// Mitsubishi GX Works2 project: PLC_Project_v156 final   PLC: FX3G

// global labels: Global1
VAR_GLOBAL
  X_0 AT X000 : BOOL;
  X_1 AT X001 : BOOL;
  X_2 AT X002 : BOOL;
  X_3 AT X003 : BOOL;
  X_4 AT X004 : BOOL;
  X_5 AT X005 : BOOL;
  X_6 AT X006 : BOOL;
  X_7 AT X007 : BOOL;
  Y_0 AT Y000 : BOOL;
  Y_1 AT Y001 : BOOL;
  Y_2 AT Y002 : BOOL;
  Y_3 AT Y003 : BOOL;
  Y_4 AT Y004 : BOOL;
  Y_5 AT Y005 : BOOL;
  Y_6 AT Y006 : BOOL;
  Y_7 AT Y007 : BOOL;
  SINGLE_POP_PACK : BOOL;
  FLVR_PRO_START : BOOL;
  COOLING_START : BOOL;
  TEMP_SENSOR : BOOL;
  PACKAGING_START : BOOL;
  EMERGENCY_BTN : BOOL;
  FACTORY_START : BOOL;
  FLVR_RUNNING : BOOL;
  COOLING_RUNNING : BOOL;
  CASE_PAC_RUNNING : BOOL;
  FACTORY_RUNNING : BOOL;
  ANALOG_1 AT D8280 : INT;
  TOTAL_BOX : INT;
  POP_COUNT AT CC1 : BOOL;
  COUNTER1 AT CC2 : BOOL;
  CN_1 AT CN1 : WORD;
  ANALOG_OUTPUT AT D8282 : INT;
  TIMER3_RUN : BOOL;
  MIXING_BLINK1 : BOOL;
  MIXING_BLINK2 : BOOL;
END_VAR

// task Task_01 (event TRUE, interval 0, priority 31): IO_MAP, MAIN

PROGRAM IO_MAP
(* structured ladder/FBD written out as ST: instructions are called as NAME(EN, inputs, outputs); _pN, _eN, _tN stand for wires *)
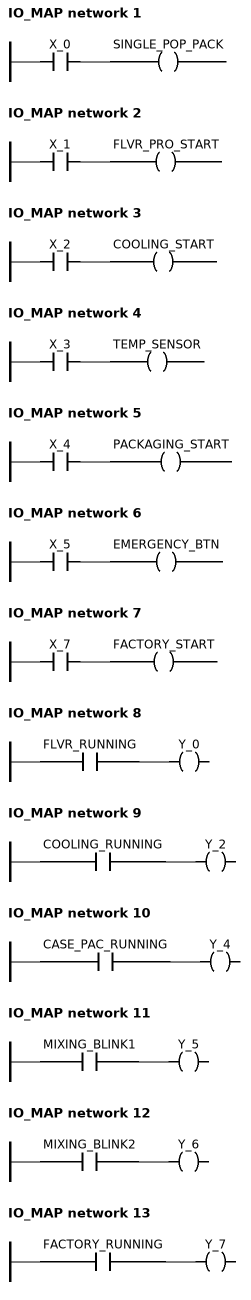
(* network 1 *)
SINGLE_POP_PACK := X_0;
(* network 2 *)
FLVR_PRO_START := X_1;
(* network 3 *)
COOLING_START := X_2;
(* network 4 *)
TEMP_SENSOR := X_3;
(* network 5 *)
PACKAGING_START := X_4;
(* network 6 *)
EMERGENCY_BTN := X_5;
(* network 7 *)
FACTORY_START := X_7;
(* network 8 *)
Y_0 := FLVR_RUNNING;
(* network 9 *)
Y_2 := COOLING_RUNNING;
(* network 10 *)
Y_4 := CASE_PAC_RUNNING;
(* network 11 *)
Y_5 := MIXING_BLINK1;
(* network 12 *)
Y_6 := MIXING_BLINK2;
(* network 13 *)
Y_7 := FACTORY_RUNNING;
END_PROGRAM

PROGRAM MAIN
VAR
  READY : BOOL;
  REGULAR_POP : BOOL;
  LARGE_POP : BOOL;
  POP_FLAVOR_SEL : BOOL;
  LEMON_FLVR : BOOL;
  RASB_FLVR : BOOL;
  LEMON_REQ_FLVR : INT;
  LEMON_REQ_POP : INT;
  TOTAL_LEMON_REQ : INT;
  TOTAL_STAB_REQ : INT;
  RASB_REQ_POP : INT;
  GUMMY_REQ_POP : INT;
  RASB_REQ_FLVR : INT;
  TOTAL_RASB_REQ : INT;
  LEMON_AVAILABLE : INT;
  RASB_AVAILABLE : INT;
  STAB_AVAILABLE : INT;
  GUMMY_AVAILABLE : INT;
  MATERIAL_AVAILABLE : BOOL;
  FLVR_READY : BOOL;
  COOLING_DONE : BOOL;
  TIMER3_PV : TIME;
  MIXING_DONE : BOOL;
  ONE_BOX_PACKED : BOOL;
  TEST1 : BOOL;
  TEST2 : BOOL;
  LEMON_READY : BOOL;
  RASB_READY : BOOL;
  STAB_READY : BOOL;
  GUMMY_READY : BOOL;
  TON_1 : TON;
  TON_2 : TON;
  TON_3 : TON;
  TON_4 : TON;
  TON_5 : TON;
END_VAR
(* structured ladder/FBD written out as ST: instructions are called as NAME(EN, inputs, outputs); _pN, _eN, _tN stand for wires *)
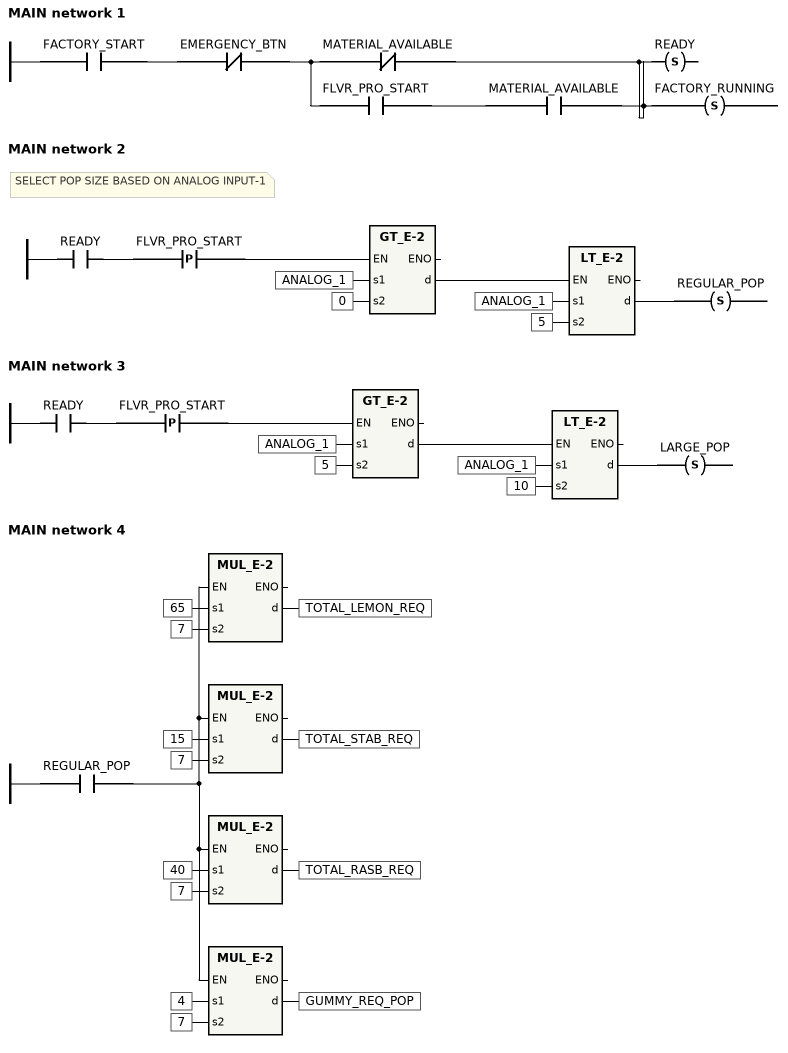
(* network 1 *)
_p1 := FACTORY_START AND NOT EMERGENCY_BTN;
_p2 := (_p1 AND NOT MATERIAL_AVAILABLE) OR (_p1 AND FLVR_PRO_START AND MATERIAL_AVAILABLE);
SET(_p2, READY);
SET(_p2, FACTORY_RUNNING);
(* network 2 *)
(* SELECT POP SIZE BASED ON ANALOG INPUT-1 *)
GT_E(READY AND LDP(TRUE, FLVR_PRO_START), ANALOG_1, 0, _t1);
LT_E(_t1, ANALOG_1, 5, _t2);
SET(_t2, REGULAR_POP);
(* network 3 *)
GT_E(READY AND LDP(TRUE, FLVR_PRO_START), ANALOG_1, 5, _t1);
LT_E(_t1, ANALOG_1, 10, _t2);
SET(_t2, LARGE_POP);
(* network 4 *)
MUL_E(REGULAR_POP, 65, 7, TOTAL_LEMON_REQ);
MUL_E(REGULAR_POP, 15, 7, TOTAL_STAB_REQ);
MUL_E(REGULAR_POP, 40, 7, TOTAL_RASB_REQ);
MUL_E(REGULAR_POP, 4, 7, GUMMY_REQ_POP);
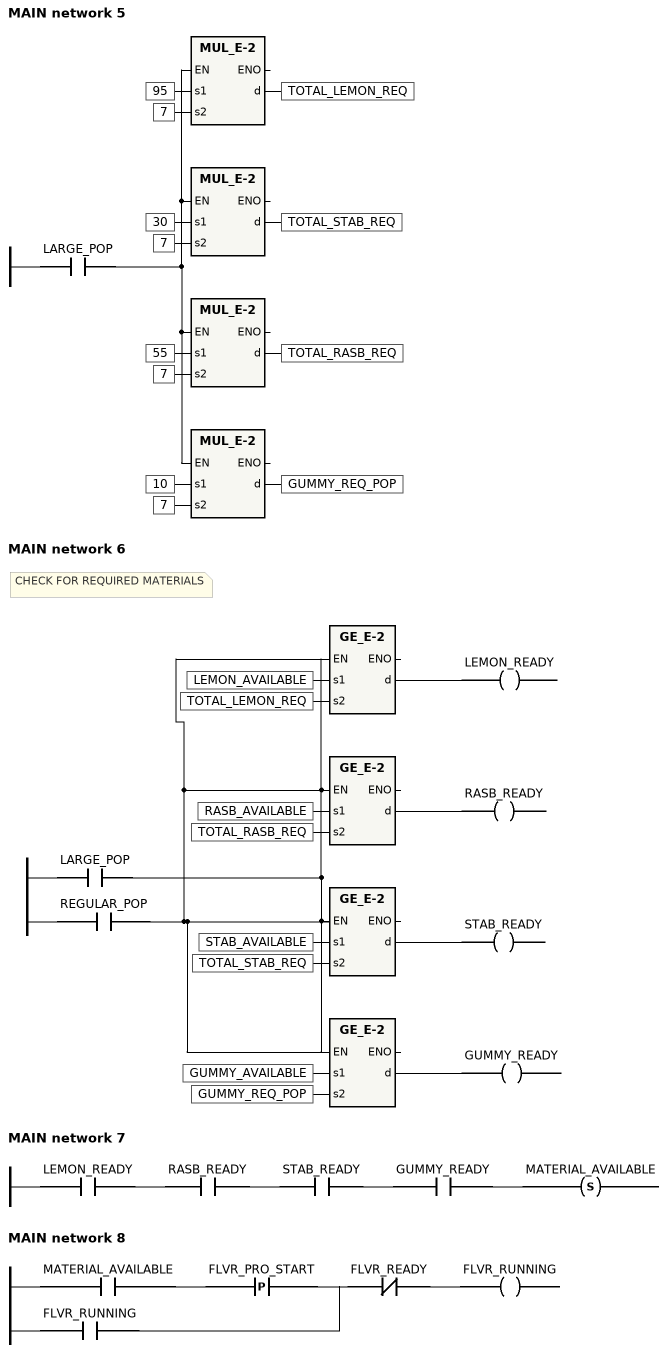
(* network 5 *)
MUL_E(LARGE_POP, 95, 7, TOTAL_LEMON_REQ);
MUL_E(LARGE_POP, 30, 7, TOTAL_STAB_REQ);
MUL_E(LARGE_POP, 55, 7, TOTAL_RASB_REQ);
MUL_E(LARGE_POP, 10, 7, GUMMY_REQ_POP);
(* network 6 *)
(* CHECK FOR REQUIRED MATERIALS *)
_p1 := LARGE_POP OR REGULAR_POP;
GE_E(_p1, LEMON_AVAILABLE, TOTAL_LEMON_REQ, _t2);
LEMON_READY := _t2;
GE_E(_p1, RASB_AVAILABLE, TOTAL_RASB_REQ, _t3);
RASB_READY := _t3;
GE_E(_p1, STAB_AVAILABLE, TOTAL_STAB_REQ, _t4);
STAB_READY := _t4;
GE_E(_p1, GUMMY_AVAILABLE, GUMMY_REQ_POP, _t5);
GUMMY_READY := _t5;
(* network 7 *)
SET(LEMON_READY AND RASB_READY AND STAB_READY AND GUMMY_READY, MATERIAL_AVAILABLE);
(* network 8 *)
FLVR_RUNNING := ((MATERIAL_AVAILABLE AND LDP(TRUE, FLVR_PRO_START)) OR FLVR_RUNNING) AND NOT FLVR_READY;
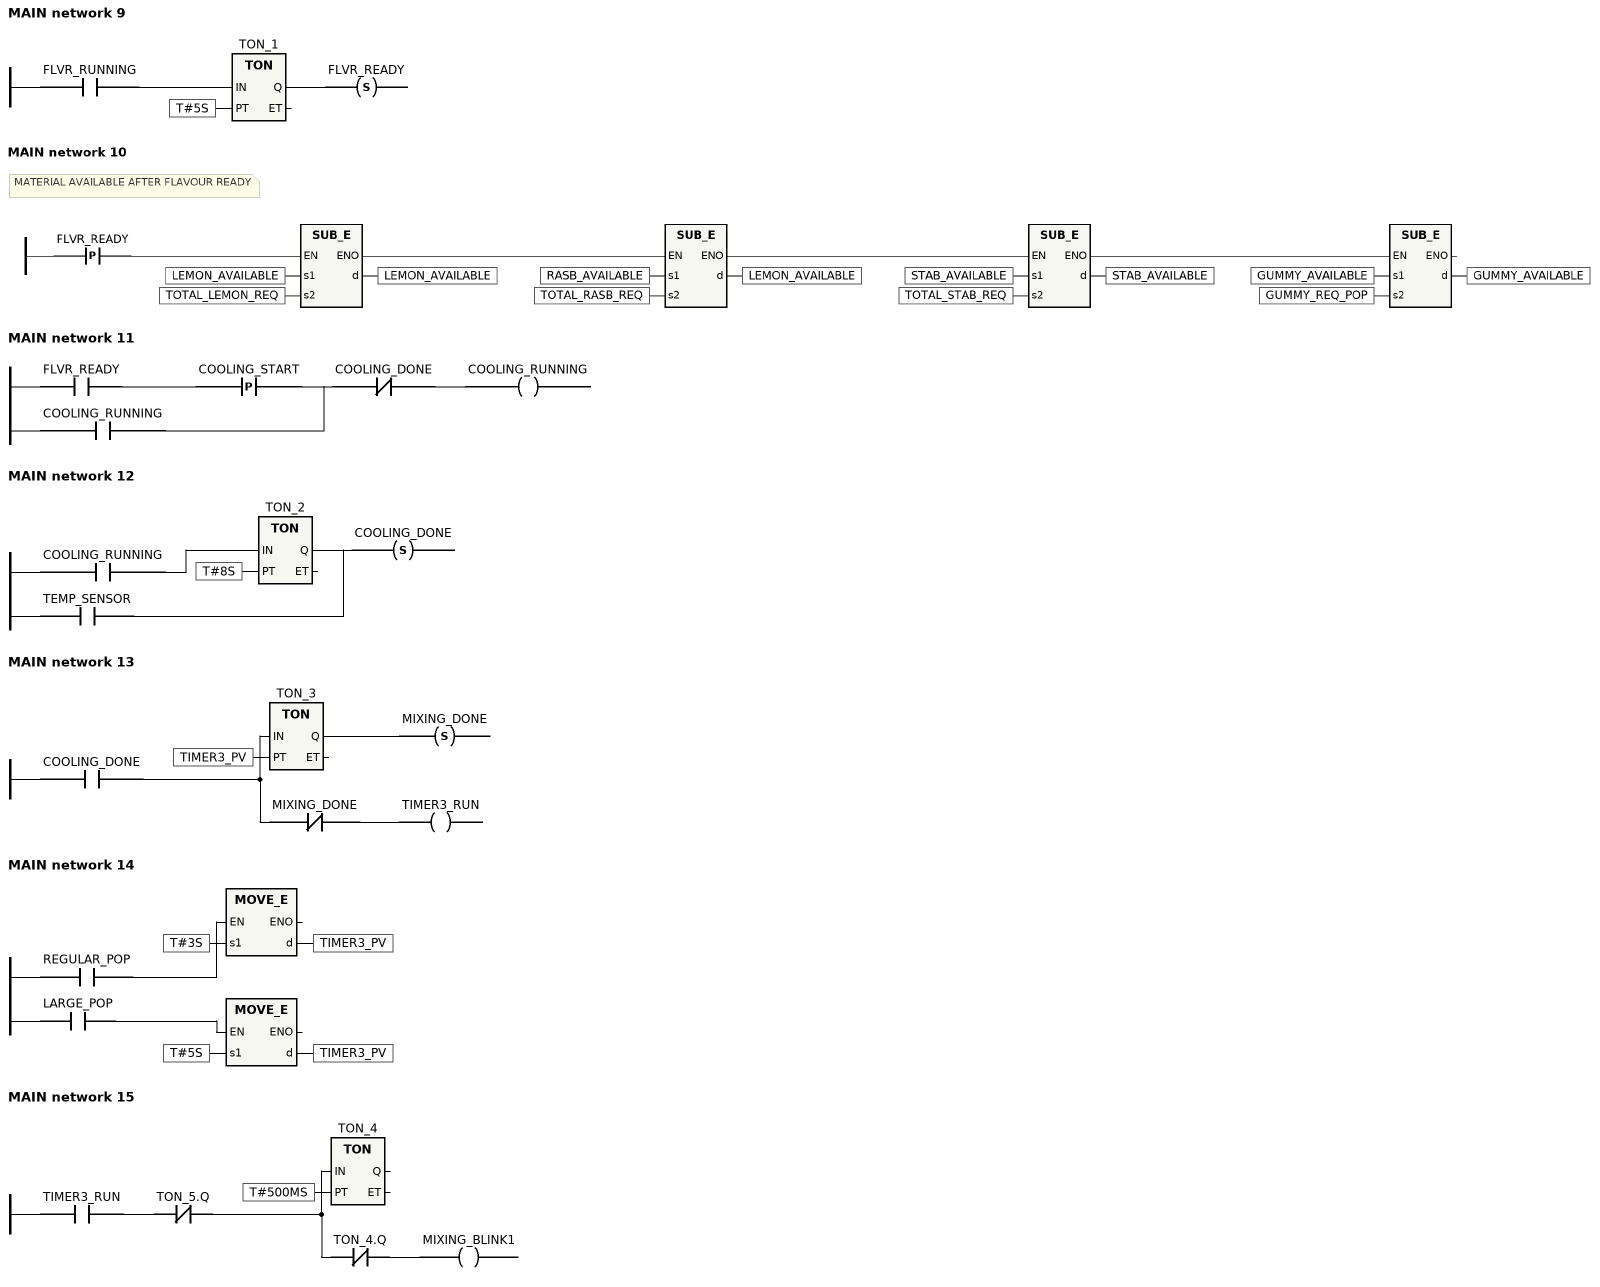
(* network 9 *)
TON_1(IN := FLVR_RUNNING, PT := T#5S);
SET(TON_1.Q, FLVR_READY);
(* network 10 *)
(* MATERIAL AVAILABLE AFTER FLAVOUR READY *)
_e1 := SUB_E(LDP(TRUE, FLVR_READY), LEMON_AVAILABLE, TOTAL_LEMON_REQ, LEMON_AVAILABLE);
_e2 := SUB_E(_e1, RASB_AVAILABLE, TOTAL_RASB_REQ, LEMON_AVAILABLE);
_e3 := SUB_E(_e2, STAB_AVAILABLE, TOTAL_STAB_REQ, STAB_AVAILABLE);
SUB_E(_e3, GUMMY_AVAILABLE, GUMMY_REQ_POP, GUMMY_AVAILABLE);
(* network 11 *)
COOLING_RUNNING := ((FLVR_READY AND LDP(TRUE, COOLING_START)) OR COOLING_RUNNING) AND NOT COOLING_DONE;
(* network 12 *)
TON_2(IN := COOLING_RUNNING, PT := T#8S);
SET(TON_2.Q OR TEMP_SENSOR, COOLING_DONE);
(* network 13 *)
TON_3(IN := COOLING_DONE, PT := TIMER3_PV);
SET(TON_3.Q, MIXING_DONE);
TIMER3_RUN := COOLING_DONE AND NOT MIXING_DONE;
(* network 14 *)
MOVE_E(REGULAR_POP, T#3S, TIMER3_PV);
MOVE_E(LARGE_POP, T#5S, TIMER3_PV);
(* network 15 *)
_p1 := TIMER3_RUN AND NOT TON_5.Q;
TON_4(IN := _p1, PT := T#500MS);
MIXING_BLINK1 := _p1 AND NOT TON_4.Q;
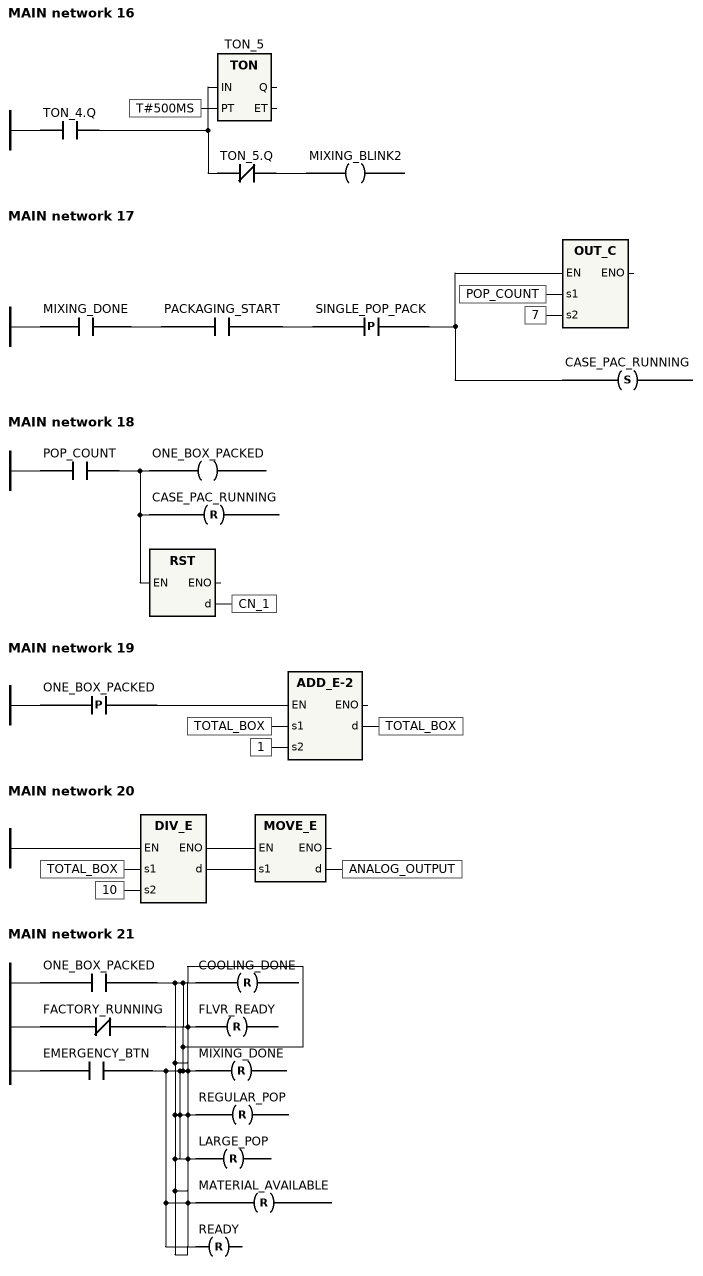
(* network 16 *)
TON_5(IN := TON_4.Q, PT := T#500MS);
MIXING_BLINK2 := TON_4.Q AND NOT TON_5.Q;
(* network 17 *)
_p1 := MIXING_DONE AND PACKAGING_START AND LDP(TRUE, SINGLE_POP_PACK);
OUT_C(_p1, POP_COUNT, 7);
SET(_p1, CASE_PAC_RUNNING);
(* network 18 *)
ONE_BOX_PACKED := POP_COUNT;
RST(POP_COUNT, CASE_PAC_RUNNING);
RST(POP_COUNT, CN_1);
(* network 19 *)
ADD_E(LDP(TRUE, ONE_BOX_PACKED), TOTAL_BOX, 1, TOTAL_BOX);
(* network 20 *)
_e2 := DIV_E(TRUE, TOTAL_BOX, 10, _t1);
MOVE_E(_e2, _t1, ANALOG_OUTPUT);
(* network 21 *)
_p1 := ONE_BOX_PACKED OR (NOT FACTORY_RUNNING) OR EMERGENCY_BTN;
RST(_p1, COOLING_DONE);
RST(_p1, FLVR_READY);
RST(_p1, MIXING_DONE);
RST(_p1, REGULAR_POP);
RST(_p1, LARGE_POP);
RST(_p1, MATERIAL_AVAILABLE);
RST(_p1, READY);
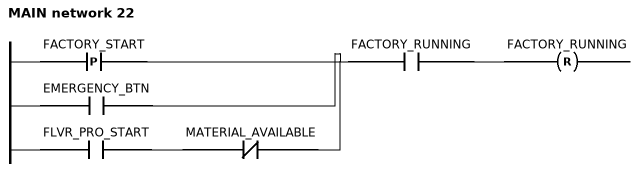
(* network 22 *)
RST((LDP(TRUE, FACTORY_START) OR EMERGENCY_BTN OR (FLVR_PRO_START AND NOT MATERIAL_AVAILABLE)) AND FACTORY_RUNNING, FACTORY_RUNNING);
END_PROGRAM
